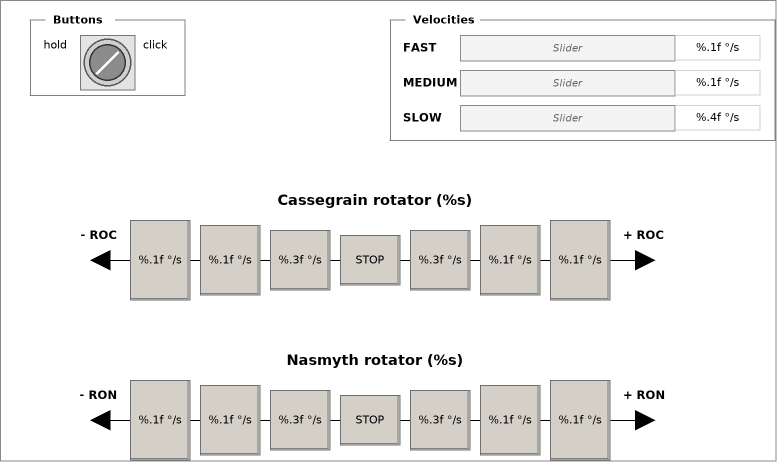
VISUALIZATION VISU_AxesManual_Joystick_Rot  // 777x462
VAR_IN_OUT
	ref : Axes;
    widget : AxesManualJoystickRotWidget;
END_VAR
    Polyline (405,20) (390,20) (390,140) (775,140) (775,20) (480,20)
    Line (110,260) (645,260)
    Slider (460,35 215x26), variable: widget.joystick_velocity_fast, input disabled if: widget.joystick_disabled, scale 0..3
    Button (270,230 60x60), "%.3f °/s", text variable: widget.joystick_velocity_slow, input disabled if: widget.jog_roc_disabled
        tap widget.jog_roc_backwards_slow
    Button (200,225 60x70), "%.1f °/s", text variable: widget.joystick_velocity_medium, input disabled if: widget.jog_roc_disabled
        tap widget.jog_roc_backwards_medium
    Button (130,220 60x80), "%.1f °/s", text variable: widget.joystick_velocity_fast, input disabled if: widget.jog_roc_disabled
        tap widget.jog_roc_backwards_fast
    Button (550,220 60x80), "%.1f °/s", text variable: widget.joystick_velocity_fast, input disabled if: widget.jog_roc_disabled
        tap widget.jog_roc_forward_fast
    Button (480,225 60x70), "%.1f °/s", text variable: widget.joystick_velocity_medium, input disabled if: widget.jog_roc_disabled
        tap widget.jog_roc_forward_medium
    Button (410,230 60x60), "%.3f °/s", text variable: widget.joystick_velocity_slow, input disabled if: widget.jog_roc_disabled
        tap widget.jog_roc_forward_slow
    Textfield (675,35 85x25), "%.1f °/s", text variable: widget.joystick_velocity_fast, input disabled if: widget.joystick_disabled
        OnMouseClick: write the text variable via VisuDialogs.Numpad, min 0, max 6
    Polygon (635,270) (635,250) (655,260)
    Polygon (110,270) (110,250) (90,260)
    Label (400,35 70x25), "FAST"
    Slider (460,70 215x26), variable: widget.joystick_velocity_medium, input disabled if: widget.joystick_disabled, scale 0..3
    Label (400,70 70x25), "MEDIUM"
    Slider (460,105 215x26), variable: widget.joystick_velocity_slow, input disabled if: widget.joystick_disabled, scale 0..3
    Label (400,105 70x25), "SLOW"
    Label (410,10 70x20), "Velocities"
    Textfield (675,70 85x25), "%.1f °/s", text variable: widget.joystick_velocity_medium, input disabled if: widget.joystick_disabled
        OnMouseClick: write the text variable via VisuDialogs.Numpad, min 0, max 3
    Textfield (675,105 85x25), "%.4f °/s", text variable: widget.joystick_velocity_slow, input disabled if: widget.joystick_disabled
        OnMouseClick: write the text variable via VisuDialogs.Numpad, min 0, max 3
    Label (620,220 45x30), "+ ROC"
    Label (80,220 40x30), "- ROC"
    Button (340,235 60x50), "STOP", input disabled if: widget.jog_roc_disabled
        OnMouseClick: execute { ref.parts.roc.processes.stop.request(); }
    Polyline (45,20) (30,20) (30,95) (185,95) (185,20) (115,20)
    RotarySwitch (80,35 55x55), variable: widget.joystick_hold, input disabled if: widget.joystick_disabled, behaviour: TOGGLE, style: Switch-RotarySwitch-Gray
    Label (140,35 50x20), "click"
    Label (30,35 40x20), "hold"
    Label (50,10 65x20), "Buttons"
    Line (110,420) (645,420)
    Button (270,390 60x60), "%.3f °/s", text variable: widget.joystick_velocity_slow, input disabled if: widget.jog_ron_disabled
        tap widget.jog_ron_backwards_slow
    Button (200,385 60x70), "%.1f °/s", text variable: widget.joystick_velocity_medium, input disabled if: widget.jog_ron_disabled
        tap widget.jog_ron_backwards_medium
    Button (130,380 60x80), "%.1f °/s", text variable: widget.joystick_velocity_fast, input disabled if: widget.jog_ron_disabled
        tap widget.jog_ron_backwards_fast
    Button (550,380 60x80), "%.1f °/s", text variable: widget.joystick_velocity_fast, input disabled if: widget.jog_ron_disabled
        tap widget.jog_ron_forward_fast
    Button (480,385 60x70), "%.1f °/s", text variable: widget.joystick_velocity_medium, input disabled if: widget.jog_ron_disabled
        tap widget.jog_ron_forward_medium
    Button (410,390 60x60), "%.3f °/s", text variable: widget.joystick_velocity_slow, input disabled if: widget.jog_ron_disabled
        tap widget.jog_ron_forward_slow
    Polygon (635,430) (635,410) (655,420)
    Polygon (110,430) (110,410) (90,420)
    Label (620,380 45x30), "+ RON"
    Label (80,380 40x30), "- RON"
    Button (340,395 60x50), "STOP", input disabled if: widget.jog_ron_disabled
        OnMouseClick: execute { ref.parts.ron.processes.stop.request(); }
    Rectangle (95,185 560x30), "Cassegrain rotator (%s)", text variable: ref.config.cassegrainRotatorName
    Rectangle (95,345 560x30), "Nasmyth rotator (%s)", text variable: ref.config.nasmythRotatorName
END_VISUALIZATION

(* stored: Version 1.1.0.1, ProductVersion 3.1.4019.2
   Visu VISU_AxesManual_Joystick_Rot: Id {277b0e0a-bc55-494e-9f73-df794e0d8cc0} *)
